// Mitsubishi GX Works2 project: 装配   PLC: FX3U/FX3UC

PROGRAM MAIN
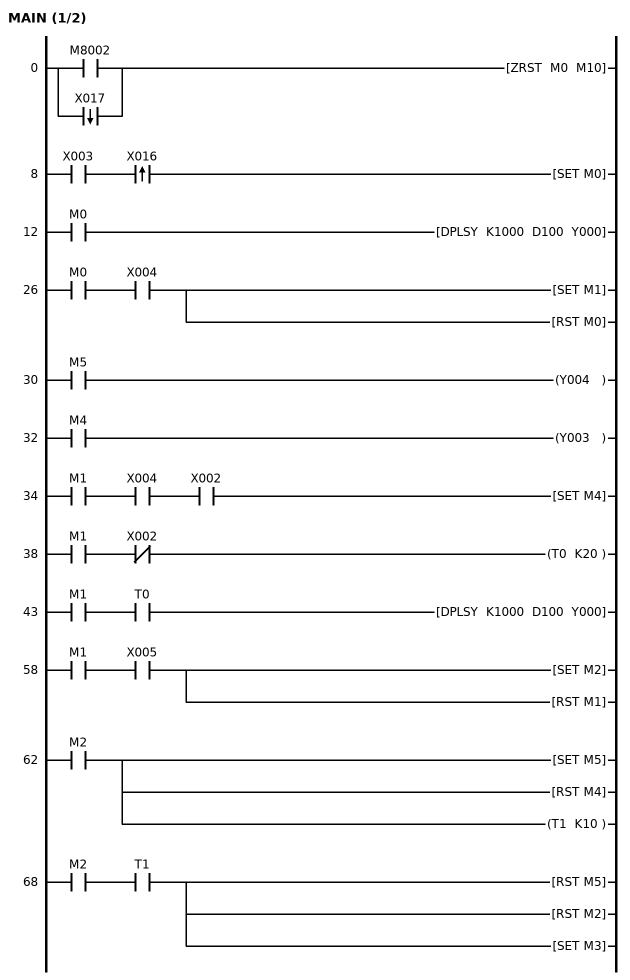
0     LD      M8002
      ORF     X017
      ZRST    M0 M10
8     LD      X003
      ANDP    X016
      SET     M0
12    LD      M0
      DPLSY   K1000 D100 Y000
26    LD      M0
      AND     X004
      SET     M1
      RST     M0
30    LD      M5
      OUT     Y004
32    LD      M4
      OUT     Y003
34    LD      M1
      AND     X004
      AND     X002
      SET     M4
38    LD      M1
      ANI     X002
      OUT     T0 K20
43    LD      M1
      AND     T0
      DPLSY   K1000 D100 Y000
58    LD      M1
      AND     X005
      SET     M2
      RST     M1
62    LD      M2
      SET     M5
      RST     M4
      OUT     T1 K10
68    LD      M2
      AND     T1
      RST     M5
      RST     M2
      SET     M3
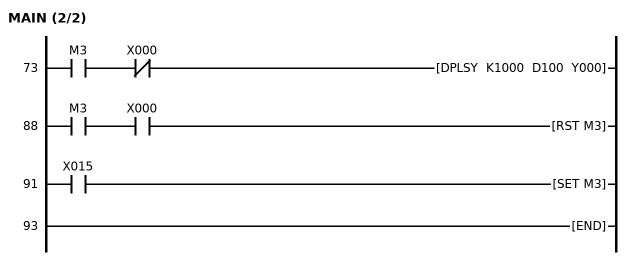
73    LD      M3
      ANI     X000
      DPLSY   K1000 D100 Y000
88    LD      M3
      AND     X000
      RST     M3
91    LD      X015
      SET     M3
93    END
END_PROGRAM
